TYPE pancake_params_0 :
STRUCT
	radius : LREAL := 100; // radius of pancake coil in mm
END_STRUCT
END_TYPE

(* stored: Version 1.1.0.1, ProductVersion 3.1.4024.12
   DUT pancake_params_0: Id {1769945b-20ab-44d0-b148-a16dfae9e3b7} *)
